Staubli VAL3: FORM_BYE.pgx

public program Form_Bye()
begin

 //程序结束界面
 cls()
 call Control_PanelMd("感谢使用史陶比尔机器人软件")



end
